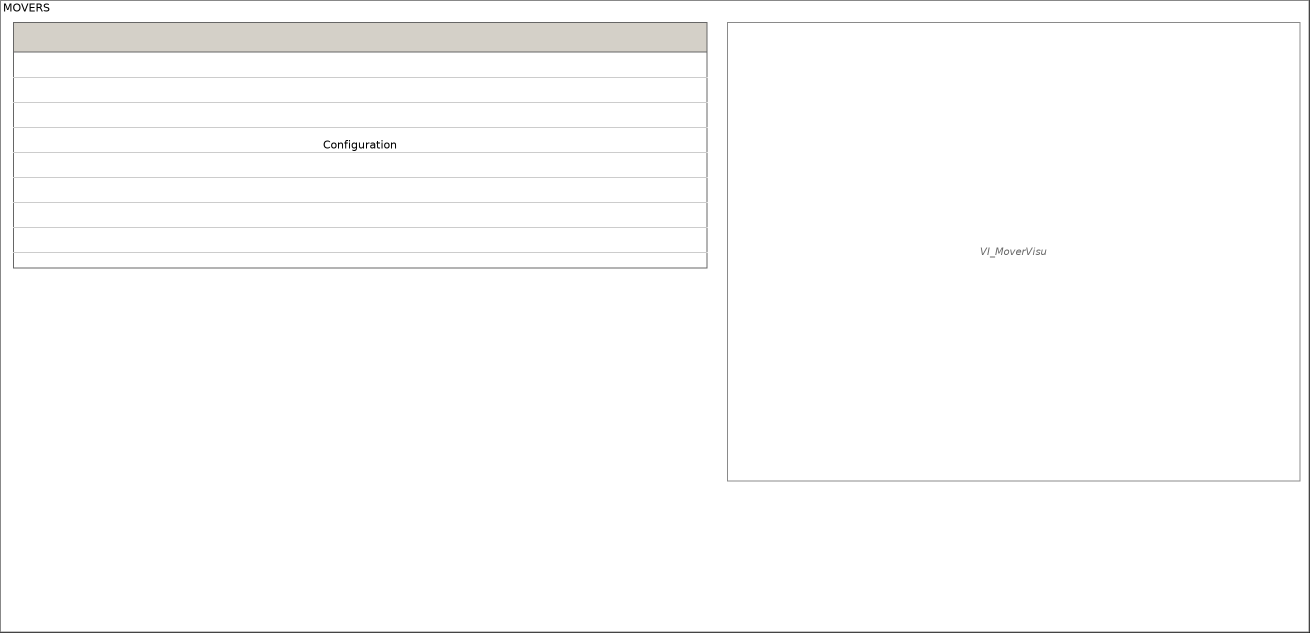
VISUALIZATION VI_MoversVisu  // 1310x633
VAR_IN_OUT
	ax		: ARRAY [1..Tc3_XTS_Utility.TcIoXtsEnvironmentParameterList.MaxXtsMoversPerXpu] OF FB_Mover;
END_VAR
VAR
	stTableStruct : ARRAY [1..25] OF stTableStructx10;
	iSelectedMover : INT;
END_VAR
    Rectangle (0,0 1310x633), "MOVERS"
    Frame (727,22 573x459), frame switch variable: iSelectedMover-1
        shows VI_MoverVisu(fbMover := ax[1])
        shows VI_MoverVisu(fbMover := ax[2])
        shows VI_MoverVisu(fbMover := ax[3])
        shows VI_MoverVisu(fbMover := ax[4])
        shows VI_MoverVisu(fbMover := ax[5])
        shows VI_MoverVisu(fbMover := ax[6])
        shows VI_MoverVisu(fbMover := ax[7])
        shows VI_MoverVisu(fbMover := ax[8])
        shows VI_MoverVisu(fbMover := ax[9])
        shows VI_MoverVisu(fbMover := ax[10])
        shows VI_MoverVisu(fbMover := ax[11])
        shows VI_MoverVisu(fbMover := ax[12])
        shows VI_MoverVisu(fbMover := ax[13])
        shows VI_MoverVisu(fbMover := ax[14])
        shows VI_MoverVisu(fbMover := ax[15])
        shows VI_MoverVisu(fbMover := ax[16])
        shows VI_MoverVisu(fbMover := ax[17])
        shows VI_MoverVisu(fbMover := ax[18])
        shows VI_MoverVisu(fbMover := ax[19])
        shows VI_MoverVisu(fbMover := ax[20])
        shows VI_MoverVisu(fbMover := ax[21])
        shows VI_MoverVisu(fbMover := ax[22])
        shows VI_MoverVisu(fbMover := ax[23])
        shows VI_MoverVisu(fbMover := ax[24])
        shows VI_MoverVisu(fbMover := ax[25])
    Table (13,22 694x246), "Configuration", data array: stTableStruct
        p1137915858: iSelectedMover
        p3854506369: ax[INDEX].ax.NcToPlc.AxisId
        p1892666644: ax[INDEX].ax.NcToPlc.ModuloSetPos
        p338671338: ax[INDEX].ax.NcToPlc.SetVelo
        p2170511999: ax[INDEX].ax.Status.MotionState
        p3723444502: ax[INDEX].ax.NcToPlc.ErrorCode
        p511219082: Position
        p1755163831: Velocity
        p2237128397: Error ID
        p505689113: Process Time
        p1757482276: Stop Positions
        p4088588272: Ack Mode
        p2243050616: Disable
        p516019884: Travel Time
        p2685023577: stTableStruct.b1
        p3312258591: stTableStruct.b2
        p1791247317: stTableStruct.b3
        p262371475: stTableStruct.b4
        p4008173056: stTableStruct.b5
        p2340480326: stTableStruct.b6
        p606709900: stTableStruct.b7
        p1095668682: stTableStruct.b8
        p1037165547: stTableStruct.b9
        p1488378029: stTableStruct.b10
        Columns.Column.[8].Template: xts.aStations[INDEX].stCfg.bDisable=true; toggle xts.aStations[INDEX].stCfg.bDisable
        Columns.Column.[6].Template: OnMouseClick: write the text variable via Default, min 1, max 3
        Columns.Column.[4].Template: OnMouseClick: write the text variable via Default
        Columns.Column.[5].Template: OnMouseClick: write the text variable via Default
        Columns.Column.[7].Template: OnMouseClick: write the text variable via Default
        Columns.Column.[9].Template: OnMouseClick: write the text variable via Default
END_VISUALIZATION

(* stored: Version 1.1.0.1, ProductVersion 3.1.4024.11
   Visu VI_MoversVisu: Id {6721de8a-7d16-4d95-a4eb-01620a6488ab} *)
